FUNCTION_BLOCK FB_SafetyBase
VAR_INPUT
END_VAR
VAR_OUTPUT
	eCurrentState : E_SafetyState;
END_VAR
VAR
END_VAR

eCurrentState := E_SafetyState.Locked;

METHOD M_Control : ERRORID
VAR_INPUT
	eCtrl : E_SafetyCtrl;
END_VAR
END_METHOD

METHOD M_MesBoxOn : ERRORID
VAR_INPUT
END_VAR
END_METHOD

END_FUNCTION_BLOCK

(* stored: Version 1.1.0.1, ProductVersion 3.1.4022.12
   POU FB_SafetyBase: Id {b5db477d-5c7e-44a0-92a7-31f4293dad49}, SpecialFunc None
   Method M_Control: Id {cb601563-1aae-4609-92ad-51b4ca46df86}
   Method M_MesBoxOn: Id {22cf7d7f-4f32-4f1c-b8bc-902214350d0c} *)
